Yaskawa INFORM job: TOOL.JBI

/JOB
//NAME TOOL
//POS
///NPOS 7,0,0,0,0,0
///TOOL 1
///POSTYPE PULSE
///PULSE
C00000=48106,30844,-23797,6986,-36730,-5014
C00001=11558,53001,-63794,-111271,-74513,80296
C00002=18930,96938,29919,-52209,-91474,35965
C00003=74585,32241,-64122,107165,-52272,-55368
C00004=75485,120600,39542,62831,-103916,-15078
C00005=46938,88554,47777,2180,-85780,-1352
C00006=75577,90930,14874,53017,-86572,27140
//INST
///DATE 2023/09/22 08:53
///ATTR SC,RW
///GROUP1 RB1
NOP
MOVJ C00000
MOVJ C00001
MOVJ C00002
MOVJ C00003
MOVJ C00004
MOVJ C00005
MOVJ C00006
END
